FUNCTION_BLOCK FB_IciciBank EXTENDS FB_Bank

VAR
END_VAR

METHOD FINAL M_Deposit : BOOL
VAR_INPUT
	fDepositAmount : REAL;
END_VAR
END_METHOD

END_FUNCTION_BLOCK

(* stored: Version 1.1.0.1, ProductVersion 3.1.4024.16
   POU FB_IciciBank: Id {b3ccc089-4f38-4011-9826-7b384ddb5fc8}, SpecialFunc None
   Method M_Deposit: Id {49045053-ad4d-4328-8980-783958c75bc1} *)
